Staubli VAL3: reset.pgx

program reset()
  local num ln_task_i
begin

  // najprej ustavimo gibanje robota, pobrišemo vse naslednje gibe, ki bi se morali zgoditi in končamo vsa opravila
  taskKill("palacinka")
  taskKill("masa")
  taskKill("obrat")
  taskKill("kroznik")
  taskKill("samodejno")
  taskKill("home")
  stopMove()
  resetMotion()
  waitEndMove()
  call cakajProgress(1)

  // Ugasnili smo vse "glavne" taske, tako da lahko to spremenljivko nastavimo na 0,
  // s čimer spet dovolimo da se v taski() podprogramu naredi nov task
  nTaskWorking = 0
end
